FUNCTION_BLOCK PUBL_3_OK (* 3-variable data publisher *)
  (* Standard: 61499-2 *)
  (* Version 1.0, 21-03-12, GASR, Universidade do Estado de Santa Catarina *)
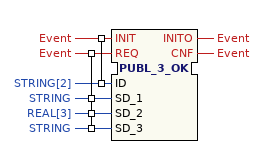
  EVENT_INPUT
    INIT WITH ID; (* Service initiaization *)
    REQ WITH SD_1, SD_2, SD_3;
  END_EVENT
  EVENT_OUTPUT
    INITO; (* Initialization Confirm *)
    CNF; (* Service confirmation *)
  END_EVENT
  VAR_INPUT
    ID : ARRAY [0..1] OF STRING; (* Default id is the FB instance name *)
    SD_1 : STRING;
    SD_2 : ARRAY [0..2] OF REAL; (* Machine Position *)
    SD_3 : STRING; (* Current tool *)
  END_VAR
  SERVICE PUBL_3_OK/SUBL_3_OK (* Data publication service *)
    SEQUENCE normal_establishment
      PUBL_3_OK.INIT(ID) -> PUBL_3_OK.INITO();
      SUBL_3_OK.INIT(ID) -> SUBL_3_OK.INITO();
    END_SEQUENCE
    SEQUENCE normal_data_transfer
      PUBL_3_OK.REQ(SD_1,SD_2,SD_3) -> SUBL_3_OK.IND(RD_1,RD_2,RD_3);
    END_SEQUENCE
  END_SERVICE
END_FUNCTION_BLOCK
